// Brief: Master Arm Initialization
FUNCTION_BLOCK PUBLIC FB_ArmStandBy EXTENDS FB_MasterArmCtrlBase
VAR_INPUT
END_VAR
VAR_OUTPUT
END_VAR
VAR
END_VAR

// override this function in each exact controller
// NOTICE: set joint control mode here, and do some initialization if needed
METHOD PROTECTED Init : BOOL
VAR_IN_OUT CONSTANT
	i_masterArm :FB_MasterArm;
	i_masterArmCtrlCmd :ST_ArmCtrlCmds;
END_VAR
VAR
	j:INT;
	maxJntErr:LREAL;
	jntCtrlErr:Vec7d;
END_VAR
SUPER^.Init(i_masterArm,i_masterArmCtrlCmd);

// check if to hold the command joint position unchanged
jntCtrlErr:=subVec7(i_masterArmCtrlCmd.m_cmdJntPos, i_masterArm.m_curJntPos);
maxJntErr:=0.0;
FOR j:=1 TO g_mJntNum DO
	maxJntErr:= MAX(maxJntErr, ABS(jntCtrlErr[j]));
END_FOR

IF maxJntErr<g_jntCtrlErrForCmdHold THEN
	m_cmdJntPos:=i_masterArmCtrlCmd.m_cmdJntPos;
ELSE
	m_cmdJntPos:=i_masterArm.curJntPos;
END_IF
END_METHOD

END_FUNCTION_BLOCK

(* stored: Version 1.1.0.1, ProductVersion 3.1.4024.12
   POU FB_ArmStandBy: Id {82e389e4-7a38-4619-a14b-0246d1236311}, SpecialFunc None
   Method Init: Id {e4eba8ef-1092-44ea-8fed-edb6d236e75a} *)
